FUNCTION_BLOCK FB_SHIFT1_DT (* Stores the input and outputs the data upon the next request *)
  (* Standard: 61499-2 *)
  (* Version 1.1, 2017-06-13, Marc Jakobi, HTW Berlin *)
  (* Version 1.0, 2016-05-26, AZ, fortiss GmbH *)
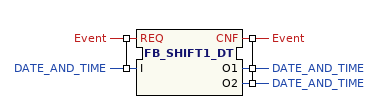
  EVENT_INPUT
    REQ WITH I; (* Normal Execution Request *)
  END_EVENT
  EVENT_OUTPUT
    CNF WITH O1, O2; (* Execution Confirmation *)
  END_EVENT
  VAR_INPUT
    I : DATE_AND_TIME; (* Input *)
  END_VAR
  VAR_OUTPUT
    O1 : DATE_AND_TIME; (* Current output *)
    O2 : DATE_AND_TIME; (* Last output (O1 of last request) *)
  END_VAR
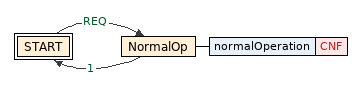
  EC_STATES
    START;
    NormalOp : normalOperation -> CNF; (* Normal execution *)
  END_STATES
  EC_TRANSITIONS
    START TO NormalOp := REQ;
    NormalOp TO START := 1;
  END_TRANSITIONS
  ALGORITHM normalOperation IN ST:
O2 := O1;
O1 := I;
  END_ALGORITHM
END_FUNCTION_BLOCK
